// TwinCAT 3 PLC project TcUnitTest
// ProgramVersion: 3.1.4024.0
// libraries:
//   Tc2_Standard, * (Beckhoff Automation GmbH)
//   Tc2_System, * (Beckhoff Automation GmbH)
//   Tc3_Module, * (Beckhoff Automation GmbH)
//   TcUnit, * (www.tcunit.org)
// project tree:
//   / PlcTask.TcTTO
//   MyLibrary/ FB_Calculator.TcPOU
//   Test/ FB_Calculator_Test.TcPOU, PRG_TEST.TcPOU
// real-time tasks:
//   TASK PlcTask: cycle T#10ms, priority 20, ADS port 350

CONFIGURATION TcUnitTest
    RESOURCE PLC ON TwinCAT3
        TASK PlcTask(INTERVAL := T#10ms, PRIORITY := 20);
        PROGRAM PRG_TEST WITH PlcTask : PRG_TEST;
    END_RESOURCE
END_CONFIGURATION

// ---- Test/PRG_TEST.TcPOU
PROGRAM PRG_TEST
VAR
	fbCalculatorTest : FB_Calculator_Test;
END_VAR

TcUnit.RUN();

END_PROGRAM

// ---- Test/FB_Calculator_Test.TcPOU
FUNCTION_BLOCK FB_Calculator_Test EXTENDS FB_TestSuite
VAR
END_VAR

AddOnePlusOneExpectTwo();
SubThreeMinusTwoExpectOne();

METHOD PRIVATE AddOnePlusOneExpectTwo : LREAL;
VAR
	fbCalculator : FB_Calculator;
	result: LREAL;
END_VAR
TEST('AddOnePlusOneExpectTwo');

	// @TEST-RUN
	result := fbCalculator.Addition(a:=1,b:=1);
	
	// @TEST-ASSERT
	AssertEquals_LREAL(Expected:=2,Actual:=result,Delta:=0.0,Message:=' Addition was not OK');
	
TEST_FINISHED();
END_METHOD

METHOD PRIVATE SubThreeMinusTwoExpectOne : LREAL
VAR
	result: LREAL;
	fbCalculator: FB_Calculator;
END_VAR
TEST('SubThreeMinusTwoExpectOne');

	// @TEST-RUN
	result := fbCalculator.Substraction(a:=3,b:=2);
	
	// @TEST-ASSERT
	AssertEquals_LREAL(Expected:=1,Actual:=result,Delta:=0.0,Message:='Substraction was not OK');
	
TEST_FINISHED();
END_METHOD

END_FUNCTION_BLOCK

// ---- MyLibrary/FB_Calculator.TcPOU
FUNCTION_BLOCK FB_Calculator
VAR
END_VAR

METHOD Addition : LREAL;
VAR_INPUT
	a : LREAL;
	b : LREAL;
END_VAR
Addition := a + b;
END_METHOD

METHOD Substraction : LREAL
VAR_INPUT
	a : LREAL;
	b : LREAL;
END_VAR
Substraction := a - b;
END_METHOD

END_FUNCTION_BLOCK
